// TIA Portal V20 export
DATA_BLOCK "SafetyDoorInterface"   // DB179
// stored: Access Published, MemoryReserve 100
   VAR
      fDoor11Interface { S7_SetPoint := 'True'} : "LER_typefDoorInterface";
      fDoor10Interface { S7_SetPoint := 'True'} : "LER_typefDoorInterface";
      fDoor9Interface { S7_SetPoint := 'True'} : "LER_typefDoorInterface";
      fDoor8Interface { S7_SetPoint := 'True'} : "LER_typefDoorInterface";
      fDoor7Interface { S7_SetPoint := 'True'} : "LER_typefDoorInterface";
      fDoor6Interface { S7_SetPoint := 'True'} : "LER_typefDoorInterface";
      fDoor5Interface { S7_SetPoint := 'True'} : "LER_typefDoorInterface";
      fDoor4Interface { S7_SetPoint := 'True'} : "LER_typefDoorInterface";
      fDoor3Interface { S7_SetPoint := 'True'} : "LER_typefDoorInterface";
      fDoor2Interface { S7_SetPoint := 'True'} : "LER_typefDoorInterface";
      fDoor1Interface { S7_SetPoint := 'True'} : "LER_typefDoorInterface";
      TON { S7_SetPoint := 'True'} : Array[0..9] of TON_TIME;
   END_VAR
BEGIN
   fDoor11Interface.configuration.referenceDesignator := WSTRING#'MAINT';
   fDoor10Interface.configuration.referenceDesignator := WSTRING#'STK1';
   fDoor9Interface.configuration.referenceDesignator := WSTRING#'STK2';
   fDoor8Interface.configuration.referenceDesignator := WSTRING#'TR.PP L';
   fDoor7Interface.configuration.referenceDesignator := WSTRING#'TR.PP';
   fDoor6Interface.configuration.referenceDesignator := WSTRING#'UNLOAD';
   fDoor5Interface.configuration.referenceDesignator := WSTRING#'WEIGHT';
   fDoor4Interface.configuration.referenceDesignator := WSTRING#'LASER';
   fDoor3Interface.configuration.referenceDesignator := WSTRING#'H.PRESS';
   fDoor2Interface.configuration.referenceDesignator := WSTRING#'S.TAPE';
   fDoor1Interface.configuration.referenceDesignator := WSTRING#'T.TAPE';
END_DATA_BLOCK
